// TIA Portal V20 export
TYPE "LER_typeCommunicationSpecialFunctions"
// stored: Access Published
   STRUCT
      specialFunction1 : Bool;
      specialFunction2 : Bool;
      specialFunction3 : Bool;
      specialFunction4 : Bool;
      specialFunction5 : Bool;
      specialFunction6 : Bool;
      specialFunction7 : Bool;
      specialFunction8 : Bool;
      specialFunction9 : Bool;
      specialFunction10 : Bool;
      specialFunction11 : Bool;
      specialFunction12 : Bool;
      specialFunction13 : Bool;
      specialFunction14 : Bool;
      specialFunction15 : Bool;
      specialFunction16 : Bool;
      specialFunction17 : Bool;
      specialFunction18 : Bool;
      specialFunction19 : Bool;
      specialFunction20 : Bool;
      specialFunction21 : Bool;
      specialFunction22 : Bool;
      specialFunction23 : Bool;
      specialFunction24 : Bool;
      specialFunction25 : Bool;
      specialFunction26 : Bool;
      specialFunction27 : Bool;
      specialFunction28 : Bool;
      specialFunction29 : Bool;
      specialFunction30 : Bool;
      specialFunction31 : Bool;
      specialFunction32 : Bool;
   END_STRUCT;
END_TYPE
